   1:  PR[91,2] = PR[90,2] + -18.989;
   1:L PR[91] R[100]mm/sec CNT100;
   1:  PR[91,1] = PR[90,1] + -71.625;
   1:  PR[91,2] = PR[90,2] + -19.966;
   1:L PR[91] R[100]mm/sec CNT100;
   1:  PR[91,1] = PR[90,1] + -67.146;
   1:  PR[91,2] = PR[90,2] + -20.149;
   1:L PR[91] R[100]mm/sec CNT100;
   1:  PR[91,1] = PR[90,1] + -63.769;
   1:  PR[91,2] = PR[90,2] + -19.645;
   1:L PR[91] R[100]mm/sec CNT100;
   1:  PR[91,1] = PR[90,1] + -62.587;
   1:  PR[91,2] = PR[90,2] + -19.490;
   1:L PR[91] R[100]mm/sec CNT100;
   1:  PR[91,1] = PR[90,1] + -60.217;
   1:  PR[91,2] = PR[90,2] + -18.649;
   1:L PR[91] R[100]mm/sec CNT100;
   1:  PR[91,1] = PR[90,1] + -58.248;
   1:  PR[91,2] = PR[90,2] + -17.990;
   1:L PR[91] R[100]mm/sec CNT100;
   1:  PR[91,1] = PR[90,1] + -56.891;
   1:  PR[91,2] = PR[90,2] + -17.175;
   1:L PR[91] R[100]mm/sec CNT100;
   1:  PR[91,1] = PR[90,1] + -54.312;
   1:  PR[91,2] = PR[90,2] + -15.689;
   1:L PR[91] R[100]mm/sec CNT100;
   1:  PR[91,1] = PR[90,1] + -53.842;
   1:  PR[91,2] = PR[90,2] + -15.250;
   1:L PR[91] R[100]mm/sec CNT100;
   1:  PR[91,1] = PR[90,1] + -50.938;
   1:  PR[91,2] = PR[90,2] + -12.631;
   1:L PR[91] R[100]mm/sec CNT100;
   1:  PR[91,1] = PR[90,1] + -48.280;
   1:  PR[91,2] = PR[90,2] + -9.189;
   1:L PR[91] R[100]mm/sec CNT100TB   .50sec,CALL END_PUD;
   1:  PR[92] = PR[91];
   1:  PR[92,3] = PR[92,3] + 20;
   1:J PR[92] 10% FINE;
   1:  PR[91] = PR[90];
   1:  PR[91,1] = PR[90,1] + -47.207;
   1:  PR[91,2] = PR[90,2] + 7.658;
   1:  PR[91,3] = PR[90,3] + 39.195;
   1:  PR[92] = PR[91];
   1:  PR[92,3] = PR[92,3] + 20;
   1:J PR[92] 10% FINE;
   1:L PR[91] R[100]mm/sec CNT100;
   1:  CALL LASER_DRAHT_START;
   1:  PR[91,1] = PR[90,1] + -49.902;
   1:  PR[91,2] = PR[90,2] + 11.311;
   1:L PR[91] R[100]mm/sec CNT100;
   1:  PR[91,1] = PR[90,1] + -51.244;
   1:  PR[91,2] = PR[90,2] + 12.483;
   1:L PR[91] R[100]mm/sec CNT100;
   1:  PR[91,1] = PR[90,1] + -53.419;
   1:  PR[91,2] = PR[90,2] + 14.347;
   1:L PR[91] R[100]mm/sec CNT100;
   1:  PR[91,1] = PR[90,1] + -57.577;
   1:  PR[91,2] = PR[90,2] + 16.651;
   1:L PR[91] R[100]mm/sec CNT100;
   1:  PR[91,1] = PR[90,1] + -60.018;
   1:  PR[91,2] = PR[90,2] + 17.440;
   1:L PR[91] R[100]mm/sec CNT100;
   1:  PR[91,1] = PR[90,1] + -62.061;
   1:  PR[91,2] = PR[90,2] + 18.166;
   1:L PR[91] R[100]mm/sec CNT100;
   1:  PR[91,1] = PR[90,1] + -66.547;
   1:  PR[91,2] = PR[90,2] + 18.829;
   1:L PR[91] R[100]mm/sec CNT100;
   1:  PR[91,1] = PR[90,1] + -68.412;
   1:  PR[91,2] = PR[90,2] + 18.760;
   1:L PR[91] R[100]mm/sec CNT100;
   1:  PR[91,1] = PR[90,1] + -71.023;
   1:  PR[91,2] = PR[90,2] + 18.639;
   1:L PR[91] R[100]mm/sec CNT100;
   1:  PR[91,1] = PR[90,1] + -75.333;
   1:  PR[91,2] = PR[90,2] + 17.623;
   1:L PR[91] R[100]mm/sec CNT100;
   1:  PR[91,1] = PR[90,1] + -79.285;
   1:  PR[91,2] = PR[90,2] + 15.844;
   1:L PR[91] R[100]mm/sec CNT100;
   1:  PR[91,1] = PR[90,1] + -82.702;
   1:  PR[91,2] = PR[90,2] + 13.402;
   1:L PR[91] R[100]mm/sec CNT100;
   1:  PR[91,1] = PR[90,1] + -85.411;
   1:  PR[91,2] = PR[90,2] + 10.405;
   1:L PR[91] R[100]mm/sec CNT100;
   1:  PR[91,1] = PR[90,1] + -87.427;
   1:  PR[91,2] = PR[90,2] + 6.951;
   1:L PR[91] R[100]mm/sec CNT100;
   1:  PR[91,1] = PR[90,1] + -88.666;
   1:  PR[91,2] = PR[90,2] + 3.187;
   1:L PR[91] R[100]mm/sec CNT100;
   1:  PR[91,1] = PR[90,1] + -88.752;
   1:  PR[91,2] = PR[90,2] + 2.391;
   1:L PR[91] R[100]mm/sec CNT100;
   1:  PR[91,1] = PR[90,1] + -88.808;
   1:  PR[91,2] = PR[90,2] + 2.113;
   1:L PR[91] R[100]mm/sec CNT100;
   1:  PR[91,1] = PR[90,1] + -89.112;
   1:  PR[91,2] = PR[90,2] + -0.728;
   1:L PR[91] R[100]mm/sec CNT100;
   1:  PR[91,1] = PR[90,1] + -89.014;
   1:  PR[91,2] = PR[90,2] + -1.630;
   1:L PR[91] R[100]mm/sec CNT100;
   1:  PR[91,1] = PR[90,1] + -88.812;
   1:  PR[91,2] = PR[90,2] + -2.533;
   1:L PR[91] R[100]mm/sec CNT100;
   1:  PR[91,1] = PR[90,1] + -88.586;
   1:  PR[91,2] = PR[90,2] + -4.648;
   1:L PR[91] R[100]mm/sec CNT100;
   1:  PR[91,1] = PR[90,1] + -87.339;
   1:  PR[91,2] = PR[90,2] + -8.411;
   1:L PR[91] R[100]mm/sec CNT100;
   1:  PR[91,1] = PR[90,1] + -85.305;
   1:  PR[91,2] = PR[90,2] + -11.869;
   1:L PR[91] R[100]mm/sec CNT100;
   1:  PR[91,1] = PR[90,1] + -82.564;
   1:  PR[91,2] = PR[90,2] + -14.882;
   1:L PR[91] R[100]mm/sec CNT100;
   1:  PR[91,1] = PR[90,1] + -79.213;
   1:  PR[91,2] = PR[90,2] + -17.320;
   1:L PR[91] R[100]mm/sec CNT100;
   1:  PR[91,1] = PR[90,1] + -75.385;
   1:  PR[91,2] = PR[90,2] + -19.075;
   1:L PR[91] R[100]mm/sec CNT100;
   1:  PR[91,1] = PR[90,1] + -71.106;
   1:  PR[91,2] = PR[90,2] + -20.083;
   1:L PR[91] R[100]mm/sec CNT100;
   1:  PR[91,1] = PR[90,1] + -67.492;
   1:  PR[91,2] = PR[90,2] + -20.230;
   1:L PR[91] R[100]mm/sec CNT100;
   1:  PR[91,1] = PR[90,1] + -66.515;
   1:  PR[91,2] = PR[90,2] + -20.286;
   1:L PR[91] R[100]mm/sec CNT100;
   1:  PR[91,1] = PR[90,1] + -63.770;
   1:  PR[91,2] = PR[90,2] + -19.876;
   1:L PR[91] R[100]mm/sec CNT100;
   1:  PR[91,1] = PR[90,1] + -61.937;
   1:  PR[91,2] = PR[90,2] + -19.636;
   1:L PR[91] R[100]mm/sec CNT100;
   1:  PR[91,1] = PR[90,1] + -60.190;
   1:  PR[91,2] = PR[90,2] + -19.016;
   1:L PR[91] R[100]mm/sec CNT100;
   1:  PR[91,1] = PR[90,1] + -57.558;
   1:  PR[91,2] = PR[90,2] + -18.135;
   1:L PR[91] R[100]mm/sec CNT100;
   1:  PR[91,1] = PR[90,1] + -56.806;
   1:  PR[91,2] = PR[90,2] + -17.684;
   1:L PR[91] R[100]mm/sec CNT100;
   1:  PR[91,1] = PR[90,1] + -53.568;
   1:  PR[91,2] = PR[90,2] + -15.818;
   1:L PR[91] R[100]mm/sec CNT100;
   1:  PR[91,1] = PR[90,1] + -53.267;
   1:  PR[91,2] = PR[90,2] + -15.544;
   1:L PR[91] R[100]mm/sec CNT100;
   1:  PR[91,1] = PR[90,1] + -50.100;
   1:  PR[91,2] = PR[90,2] + -12.951;
   1:L PR[91] R[100]mm/sec CNT100;
   1:  PR[91,1] = PR[90,1] + -49.327;
   1:  PR[91,2] = PR[90,2] + -12.096;
   1:L PR[91] R[100]mm/sec CNT100;
   1:  PR[91,1] = PR[90,1] + -47.391;
   1:  PR[91,2] = PR[90,2] + -9.587;
   1:L PR[91] R[100]mm/sec CNT100;
   1:  PR[91,1] = PR[90,1] + -46.330;
   1:  PR[91,2] = PR[90,2] + -7.540;
   1:L PR[91] R[100]mm/sec CNT100;
   1:  PR[91,1] = PR[90,1] + -45.515;
   1:  PR[91,2] = PR[90,2] + -5.643;
   1:L PR[91] R[100]mm/sec CNT100;
   1:  PR[91,1] = PR[90,1] + -45.158;
   1:  PR[91,2] = PR[90,2] + -3.960;
   1:L PR[91] R[100]mm/sec CNT100;
   1:  PR[91,1] = PR[90,1] + -45.073;
   1:  PR[91,2] = PR[90,2] + -3.355;
   1:L PR[91] R[100]mm/sec CNT100;
   1:  PR[91,1] = PR[90,1] + -45.003;
   1:  PR[91,2] = PR[90,2] + -2.254;
   1:L PR[91] R[100]mm/sec CNT100;
   1:  PR[91,1] = PR[90,1] + -44.855;
   1:  PR[91,2] = PR[90,2] + -0.642;
   1:L PR[91] R[100]mm/sec CNT100;
   1:  PR[91,1] = PR[90,1] + -45.345;
   1:  PR[91,2] = PR[90,2] + 3.088;
   1:L PR[91] R[100]mm/sec CNT100;
   1:  PR[91,1] = PR[90,1] + -45.463;
   1:  PR[91,2] = PR[90,2] + 3.590;
   1:L PR[91] R[100]mm/sec CNT100;
   1:  PR[91,1] = PR[90,1] + -46.247;
   1:  PR[91,2] = PR[90,2] + 5.331;
   1:L PR[91] R[100]mm/sec CNT100;
   1:  PR[91,1] = PR[90,1] + -47.206;
   1:  PR[91,2] = PR[90,2] + 7.658;
   1:L PR[91] R[100]mm/sec CNT100TB   .50sec,CALL END_PUD;
   1:  PR[92] = PR[91];
   1:  PR[92,3] = PR[92,3] + 20;
   1:J PR[92] 10% FINE;
   1:  PR[91,1] = PR[90,1] + -40.199;
   1:  PR[91,2] = PR[90,2] + 4.341;
   1:  PR[92] = PR[91];
   1:  PR[92,3] = PR[92,3] + 20;
   1:J PR[92] 10% FINE;
   1:L PR[91] R[100]mm/sec CNT100;
   1:  CALL LASER_DRAHT_START;
   1:  PR[91,1] = PR[90,1] + -40.331;
   1:  PR[91,2] = PR[90,2] + 4.012;
   1:L PR[91] R[100]mm/sec CNT100;
   1:  PR[91,1] = PR[90,1] + -40.685;
   1:  PR[91,2] = PR[90,2] + 2.385;
   1:L PR[91] R[100]mm/sec CNT100;
   1:  PR[91,1] = PR[90,1] + -40.769;
   1:  PR[91,2] = PR[90,2] + 1.636;
   1:L PR[91] R[100]mm/sec CNT100;
   1:  PR[91,1] = PR[90,1] + -40.955;
   1:  PR[91,2] = PR[90,2] + -0.751;
   1:L PR[91] R[100]mm/sec CNT100;
   1:  PR[91,1] = PR[90,1] + -40.654;
   1:  PR[91,2] = PR[90,2] + -4.032;
   1:L PR[91] R[100]mm/sec CNT100;
   1:  PR[91,1] = PR[90,1] + -40.296;
   1:  PR[91,2] = PR[90,2] + -5.597;
   1:L PR[91] R[100]mm/sec CNT100;
   1:  PR[91,1] = PR[90,1] + -39.609;
   1:  PR[91,2] = PR[90,2] + -7.567;
   1:L PR[91] R[100]mm/sec CNT100;
   1:  PR[91,1] = PR[90,1] + -39.122;
   1:  PR[91,2] = PR[90,2] + -8.820;
   1:L PR[91] R[100]mm/sec CNT100;
   1:  PR[91,1] = PR[90,1] + -38.825;
   1:  PR[91,2] = PR[90,2] + -9.370;
   1:L PR[91] R[100]mm/sec CNT100;
   1:  PR[91,1] = PR[90,1] + -37.086;
   1:  PR[91,2] = PR[90,2] + -12.138;
   1:L PR[91] R[100]mm/sec CNT100;
   1:  PR[91,1] = PR[90,1] + -36.794;
   1:  PR[91,2] = PR[90,2] + -12.551;
   1:L PR[91] R[100]mm/sec CNT100;
   1:  PR[91,1] = PR[90,1] + -36.056;
   1:  PR[91,2] = PR[90,2] + -13.368;
   1:L PR[91] R[100]mm/sec CNT100;
   1:  PR[91,1] = PR[90,1] + -33.732;
   1:  PR[91,2] = PR[90,2] + -15.700;
   1:L PR[91] R[100]mm/sec CNT100;
   1:  PR[91,1] = PR[90,1] + -32.622;
   1:  PR[91,2] = PR[90,2] + -16.492;
   1:L PR[91] R[100]mm/sec CNT100;
   1:  PR[91,1] = PR[90,1] + -30.086;
   1:  PR[91,2] = PR[90,2] + -18.111;
   1:L PR[91] R[100]mm/sec CNT100;
   1:  PR[91,1] = PR[90,1] + -28.459;
   1:  PR[91,2] = PR[90,2] + -18.807;
   1:L PR[91] R[100]mm/sec CNT100;
   1:  PR[91,1] = PR[90,1] + -25.985;
   1:  PR[91,2] = PR[90,2] + -19.712;
   1:L PR[91] R[100]mm/sec CNT100;
   1:  PR[91,1] = PR[90,1] + -23.769;
   1:  PR[91,2] = PR[90,2] + -20.140;
   1:L PR[91] R[100]mm/sec CNT100;
   1:  PR[91,1] = PR[90,1] + -21.612;
   1:  PR[91,2] = PR[90,2] + -20.432;
   1:L PR[91] R[100]mm/sec CNT100;
   1:  PR[91,1] = PR[90,1] + -18.812;
   1:  PR[91,2] = PR[90,2] + -20.365;
   1:L PR[91] R[100]mm/sec CNT100;
   1:  PR[91,1] = PR[90,1] + -17.167;
   1:  PR[91,2] = PR[90,2] + -20.229;
   1:L PR[91] R[100]mm/sec CNT100;
   1:  PR[91,1] = PR[90,1] + -13.883;
   1:  PR[91,2] = PR[90,2] + -19.427;
   1:L PR[91] R[100]mm/sec CNT100;
   1:  PR[91,1] = PR[90,1] + -12.850;
   1:  PR[91,2] = PR[90,2] + -19.107;
   1:L PR[91] R[100]mm/sec CNT100;
   1:  PR[91,1] = PR[90,1] + -9.308;
   1:  PR[91,2] = PR[90,2] + -17.354;
   1:L PR[91] R[100]mm/sec CNT100;
   1:  PR[91,1] = PR[90,1] + -8.864;
   1:  PR[91,2] = PR[90,2] + -17.098;
   1:L PR[91] R[100]mm/sec CNT100;
   1:  PR[91,1] = PR[90,1] + -5.397;
   1:  PR[91,2] = PR[90,2] + -14.278;
   1:L PR[91] R[100]mm/sec CNT100;
   1:  PR[91,1] = PR[90,1] + -3.913;
   1:  PR[91,2] = PR[90,2] + -12.363;
   1:L PR[91] R[100]mm/sec CNT100;
   1:  PR[91,1] = PR[90,1] + -2.510;
   1:  PR[91,2] = PR[90,2] + -10.642;
   1:L PR[91] R[100]mm/sec CNT100;
   1:  PR[91,1] = PR[90,1] + -2.507;
   1:  PR[91,2] = PR[90,2] + -10.636;
   1:L PR[91] R[100]mm/sec CNT100;
   1:  PR[91,1] = PR[90,1] + -0.715;
   1:  PR[91,2] = PR[90,2] + -6.857;
   1:L PR[91] R[100]mm/sec CNT100;
   1:  PR[91,1] = PR[90,1] + -0.610;
   1:  PR[91,2] = PR[90,2] + -6.577;
   1:L PR[91] R[100]mm/sec CNT100;
   1:  PR[91,1] = PR[90,1] + 0.216;
   1:  PR[91,2] = PR[90,2] + -3.257;
   1:L PR[91] R[100]mm/sec CNT100;
   1:  PR[91,1] = PR[90,1] + 3.385;
   1:  PR[91,2] = PR[90,2] + -3.299;
   1:L PR[91] R[100]mm/sec CNT100;
   1:  PR[91,1] = PR[90,1] + 4.076;
   1:  PR[91,2] = PR[90,2] + -6.422;
   1:L PR[91] R[100]mm/sec CNT100;
   1:  PR[91,1] = PR[90,1] + 4.773;
   1:  PR[91,2] = PR[90,2] + -8.090;
   1:L PR[91] R[100]mm/sec CNT100;
   1:  PR[91,1] = PR[90,1] + 5.666;
   1:  PR[91,2] = PR[90,2] + -10.320;
   1:L PR[91] R[100]mm/sec CNT100;
   1:  PR[91,1] = PR[90,1] + 6.034;
   1:  PR[91,2] = PR[90,2] + -11.054;
   1:L PR[91] R[100]mm/sec CNT100;
   1:  PR[91,1] = PR[90,1] + 8.671;
   1:  PR[91,2] = PR[90,2] + -14.460;
   1:L PR[91] R[100]mm/sec CNT100;
   1:  PR[91,1] = PR[90,1] + 8.949;
   1:  PR[91,2] = PR[90,2] + -14.860;
   1:L PR[91] R[100]mm/sec CNT100;
   1:  PR[91,1] = PR[90,1] + 9.487;
   1:  PR[91,2] = PR[90,2] + -15.427;
   1:L PR[91] R[100]mm/sec CNT100;
   1:  PR[91,1] = PR[90,1] + 13.137;
   1:  PR[91,2] = PR[90,2] + -18.194;
   1:L PR[91] R[100]mm/sec CNT100;
   1:  PR[91,1] = PR[90,1] + 13.723;
   1:  PR[91,2] = PR[90,2] + -18.559;
   1:L PR[91] R[100]mm/sec CNT100;
   1:  PR[91,1] = PR[90,1] + 18.095;
   1:  PR[91,2] = PR[90,2] + -20.344;
   1:L PR[91] R[100]mm/sec CNT100;
   1:  PR[91,1] = PR[90,1] + 18.615;
   1:  PR[91,2] = PR[90,2] + -20.509;
   1:L PR[91] R[100]mm/sec CNT100;
   1:  PR[91,1] = PR[90,1] + 23.451;
   1:  PR[91,2] = PR[90,2] + -21.128;
   1:L PR[91] R[100]mm/sec CNT100;
   1:  PR[91,1] = PR[90,1] + 23.842;
   1:  PR[91,2] = PR[90,2] + -21.151;
   1:L PR[91] R[100]mm/sec CNT100;
   1:  PR[91,1] = PR[90,1] + 28.822;
   1:  PR[91,2] = PR[90,2] + -20.487;
   1:L PR[91] R[100]mm/sec CNT100;
   1:  PR[91,1] = PR[90,1] + 29.059;
   1:  PR[91,2] = PR[90,2] + -20.442;
   1:L PR[91] R[100]mm/sec CNT100;
   1:  PR[91,1] = PR[90,1] + 33.829;
   1:  PR[91,2] = PR[90,2] + -18.475;
   1:L PR[91] R[100]mm/sec CNT100;
   1:  PR[91,1] = PR[90,1] + 33.923;
   1:  PR[91,2] = PR[90,2] + -18.431;
   1:L PR[91] R[100]mm/sec CNT100;
   1:  PR[91,1] = PR[90,1] + 38.131;
   1:  PR[91,2] = PR[90,2] + -15.244;
   1:L PR[91] R[100]mm/sec CNT100;
   1:  PR[91,1] = PR[90,1] + 38.658;
   1:  PR[91,2] = PR[90,2] + -14.617;
   1:L PR[91] R[100]mm/sec CNT100;
   1:  PR[91,1] = PR[90,1] + 42.705;
   1:  PR[91,2] = PR[90,2] + -9.418;
   1:L PR[91] R[100]mm/sec CNT100;
   1:  PR[91,1] = PR[90,1] + 47.189;
   1:  PR[91,2] = PR[90,2] + -14.100;
   1:L PR[91] R[100]mm/sec CNT100;
   1:  PR[91,1] = PR[90,1] + 47.481;
   1:  PR[91,2] = PR[90,2] + -14.437;
   1:L PR[91] R[100]mm/sec CNT100;
   1:  PR[91,1] = PR[90,1] + 50.974;
   1:  PR[91,2] = PR[90,2] + -16.993;
   1:L PR[91] R[100]mm/sec CNT100;
   1:  PR[91,1] = PR[90,1] + 52.879;
   1:  PR[91,2] = PR[90,2] + -18.168;
   1:L PR[91] R[100]mm/sec CNT100;
   1:  PR[91,1] = PR[90,1] + 55.023;
   1:  PR[91,2] = PR[90,2] + -19.106;
   1:L PR[91] R[100]mm/sec CNT100;
   1:  PR[91,1] = PR[90,1] + 59.619;
   1:  PR[91,2] = PR[90,2] + -20.650;
   1:L PR[91] R[100]mm/sec CNT100;
   1:  PR[91,1] = PR[90,1] + 59.641;
   1:  PR[91,2] = PR[90,2] + -20.654;
   1:L PR[91] R[100]mm/sec CNT100;
   1:  PR[91,1] = PR[90,1] + 60.098;
   1:  PR[91,2] = PR[90,2] + -20.706;
   1:L PR[91] R[100]mm/sec CNT100;
   1:  PR[91,1] = PR[90,1] + 64.803;
   1:  PR[91,2] = PR[90,2] + -21.406;
   1:L PR[91] R[100]mm/sec CNT100;
   1:  PR[91,1] = PR[90,1] + 66.209;
   1:  PR[91,2] = PR[90,2] + -21.457;
   1:L PR[91] R[100]mm/sec CNT100;
   1:  PR[91,1] = PR[90,1] + 69.518;
   1:  PR[91,2] = PR[90,2] + -21.226;
   1:L PR[91] R[100]mm/sec CNT100;
   1:  PR[91,1] = PR[90,1] + 72.304;
   1:  PR[91,2] = PR[90,2] + -20.762;
   1:L PR[91] R[100]mm/sec CNT100;
   1:  PR[91,1] = PR[90,1] + 73.960;
   1:  PR[91,2] = PR[90,2] + -20.276;
   1:L PR[91] R[100]mm/sec CNT100;
   1:  PR[91,1] = PR[90,1] + 77.569;
   1:  PR[91,2] = PR[90,2] + -18.895;
   1:L PR[91] R[100]mm/sec CNT100;
   1:  PR[91,1] = PR[90,1] + 78.035;
   1:  PR[91,2] = PR[90,2] + -18.638;
   1:L PR[91] R[100]mm/sec CNT100;
   1:  PR[91,1] = PR[90,1] + 81.794;
   1:  PR[91,2] = PR[90,2] + -16.221;
   1:L PR[91] R[100]mm/sec CNT100;
   1:  PR[91,1] = PR[90,1] + 84.969;
   1:  PR[91,2] = PR[90,2] + -12.992;
   1:L PR[91] R[100]mm/sec CNT100;
   1:  PR[91,1] = PR[90,1] + 87.334;
   1:  PR[91,2] = PR[90,2] + -9.214;
   1:L PR[91] R[100]mm/sec CNT100;
   1:  PR[91,1] = PR[90,1] + 88.789;
   1:  PR[91,2] = PR[90,2] + -5.064;
   1:L PR[91] R[100]mm/sec CNT100;
   1:  PR[91,1] = PR[90,1] + 89.281;
   1:  PR[91,2] = PR[90,2] + -0.729;
   1:L PR[91] R[100]mm/sec CNT100;
   1:  PR[91,1] = PR[90,1] + 88.789;
   1:  PR[91,2] = PR[90,2] + 3.606;
   1:L PR[91] R[100]mm/sec CNT100;
   1:  PR[91,1] = PR[90,1] + 87.334;
   1:  PR[91,2] = PR[90,2] + 7.755;
   1:L PR[91] R[100]mm/sec CNT100;
   1:  PR[91,1] = PR[90,1] + 84.969;
   1:  PR[91,2] = PR[90,2] + 11.533;
   1:L PR[91] R[100]mm/sec CNT100;
   1:  PR[91,1] = PR[90,1] + 81.794;
   1:  PR[91,2] = PR[90,2] + 14.762;
   1:L PR[91] R[100]mm/sec CNT100;
   1:  PR[91,1] = PR[90,1] + 78.035;
   1:  PR[91,2] = PR[90,2] + 17.179;
   1:L PR[91] R[100]mm/sec CNT100;
   1:  PR[91,1] = PR[90,1] + 77.569;
   1:  PR[91,2] = PR[90,2] + 17.436;
   1:L PR[91] R[100]mm/sec CNT100;
   1:  PR[91,1] = PR[90,1] + 73.960;
   1:  PR[91,2] = PR[90,2] + 18.817;
   1:L PR[91] R[100]mm/sec CNT100;
   1:  PR[91,1] = PR[90,1] + 72.304;
   1:  PR[91,2] = PR[90,2] + 19.303;
   1:L PR[91] R[100]mm/sec CNT100;
   1:  PR[91,1] = PR[90,1] + 69.518;
   1:  PR[91,2] = PR[90,2] + 19.767;
   1:L PR[91] R[100]mm/sec CNT100;
   1:  PR[91,1] = PR[90,1] + 66.210;
   1:  PR[91,2] = PR[90,2] + 19.998;
   1:L PR[91] R[100]mm/sec CNT100;
   1:  PR[91,1] = PR[90,1] + 64.803;
   1:  PR[91,2] = PR[90,2] + 19.947;
   1:L PR[91] R[100]mm/sec CNT100;
   1:  PR[91,1] = PR[90,1] + 60.098;
   1:  PR[91,2] = PR[90,2] + 19.247;
   1:L PR[91] R[100]mm/sec CNT100;
   1:  PR[91,1] = PR[90,1] + 59.643;
   1:  PR[91,2] = PR[90,2] + 19.196;
   1:L PR[91] R[100]mm/sec CNT100;
   1:  PR[91,1] = PR[90,1] + 59.618;
   1:  PR[91,2] = PR[90,2] + 19.191;
   1:L PR[91] R[100]mm/sec CNT100;
   1:  PR[91,1] = PR[90,1] + 55.003;
   1:  PR[91,2] = PR[90,2] + 17.641;
   1:L PR[91] R[100]mm/sec CNT100;
   1:  PR[91,1] = PR[90,1] + 52.828;
   1:  PR[91,2] = PR[90,2] + 16.681;
   1:L PR[91] R[100]mm/sec CNT100;
   1:  PR[91,1] = PR[90,1] + 50.931;
   1:  PR[91,2] = PR[90,2] + 15.513;
   1:L PR[91] R[100]mm/sec CNT100;
   1:  PR[91,1] = PR[90,1] + 47.400;
   1:  PR[91,2] = PR[90,2] + 12.904;
   1:L PR[91] R[100]mm/sec CNT100;
   1:  PR[91,1] = PR[90,1] + 47.207;
   1:  PR[91,2] = PR[90,2] + 12.680;
   1:L PR[91] R[100]mm/sec CNT100;
   1:  PR[91,1] = PR[90,1] + 42.713;
   1:  PR[91,2] = PR[90,2] + 7.937;
   1:L PR[91] R[100]mm/sec CNT100;
   1:  PR[91,1] = PR[90,1] + 38.150;
   1:  PR[91,2] = PR[90,2] + 13.761;
   1:L PR[91] R[100]mm/sec CNT100;
   1:  PR[91,1] = PR[90,1] + 38.071;
   1:  PR[91,2] = PR[90,2] + 13.839;
   1:L PR[91] R[100]mm/sec CNT100;
   1:  PR[91,1] = PR[90,1] + 33.925;
   1:  PR[91,2] = PR[90,2] + 16.974;
   1:L PR[91] R[100]mm/sec CNT100;
   1:  PR[91,1] = PR[90,1] + 33.918;
   1:  PR[91,2] = PR[90,2] + 16.979;
   1:L PR[91] R[100]mm/sec CNT100;
   1:  PR[91,1] = PR[90,1] + 33.792;
   1:  PR[91,2] = PR[90,2] + 17.038;
   1:L PR[91] R[100]mm/sec CNT100;
   1:  PR[91,1] = PR[90,1] + 29.024;
   1:  PR[91,2] = PR[90,2] + 18.992;
   1:L PR[91] R[100]mm/sec CNT100;
   1:  PR[91,1] = PR[90,1] + 28.786;
   1:  PR[91,2] = PR[90,2] + 19.038;
   1:L PR[91] R[100]mm/sec CNT100;
   1:  PR[91,1] = PR[90,1] + 23.812;
   1:  PR[91,2] = PR[90,2] + 19.692;
   1:L PR[91] R[100]mm/sec CNT100;
   1:  PR[91,1] = PR[90,1] + 23.421;
   1:  PR[91,2] = PR[90,2] + 19.670;
   1:L PR[91] R[100]mm/sec CNT100;
   1:  PR[91,1] = PR[90,1] + 18.592;
   1:  PR[91,2] = PR[90,2] + 19.044;
   1:L PR[91] R[100]mm/sec CNT100;
   1:  PR[91,1] = PR[90,1] + 18.072;
   1:  PR[91,2] = PR[90,2] + 18.880;
   1:L PR[91] R[100]mm/sec CNT100;
   1:  PR[91,1] = PR[90,1] + 13.707;
   1:  PR[91,2] = PR[90,2] + 17.092;
   1:L PR[91] R[100]mm/sec CNT100;
   1:  PR[91,1] = PR[90,1] + 13.121;
   1:  PR[91,2] = PR[90,2] + 16.727;
   1:L PR[91] R[100]mm/sec CNT100;
   1:  PR[91,1] = PR[90,1] + 9.478;
   1:  PR[91,2] = PR[90,2] + 13.959;
   1:L PR[91] R[100]mm/sec CNT100;
   1:  PR[91,1] = PR[90,1] + 8.904;
   1:  PR[91,2] = PR[90,2] + 13.356;
   1:L PR[91] R[100]mm/sec CNT100;
   1:  PR[91,1] = PR[90,1] + 6.144;
   1:  PR[91,2] = PR[90,2] + 9.789;
   1:L PR[91] R[100]mm/sec CNT100;
   1:  PR[91,1] = PR[90,1] + 6.104;
   1:  PR[91,2] = PR[90,2] + 9.727;
   1:L PR[91] R[100]mm/sec CNT100;
   1:  PR[91,1] = PR[90,1] + 5.769;
   1:  PR[91,2] = PR[90,2] + 9.085;
   1:L PR[91] R[100]mm/sec CNT100;
   1:  PR[91,1] = PR[90,1] + 4.383;
   1:  PR[91,2] = PR[90,2] + 5.768;
   1:L PR[91] R[100]mm/sec CNT100;
   1:  PR[91,1] = PR[90,1] + 4.103;
   1:  PR[91,2] = PR[90,2] + 5.061;
   1:L PR[91] R[100]mm/sec CNT100;
   1:  PR[91,1] = PR[90,1] + 3.380;
   1:  PR[91,2] = PR[90,2] + 1.835;
   1:L PR[91] R[100]mm/sec CNT100;
   1:  PR[91,1] = PR[90,1] + 0.218;
   1:  PR[91,2] = PR[90,2] + 1.796;
   1:L PR[91] R[100]mm/sec CNT100;
   1:  PR[91,1] = PR[90,1] + -0.605;
   1:  PR[91,2] = PR[90,2] + 5.086;
   1:L PR[91] R[100]mm/sec CNT100;
   1:  PR[91,1] = PR[90,1] + -2.193;
   1:  PR[91,2] = PR[90,2] + 8.477;
   1:L PR[91] R[100]mm/sec CNT100;
   1:  PR[91,1] = PR[90,1] + -2.509;
   1:  PR[91,2] = PR[90,2] + 9.179;
   1:L PR[91] R[100]mm/sec CNT100;
   1:  PR[91,1] = PR[90,1] + -3.914;
   1:  PR[91,2] = PR[90,2] + 10.905;
   1:L PR[91] R[100]mm/sec CNT100;
   1:  PR[91,1] = PR[90,1] + -5.385;
   1:  PR[91,2] = PR[90,2] + 12.808;
   1:L PR[91] R[100]mm/sec CNT100;
   1:  PR[91,1] = PR[90,1] + -8.852;
   1:  PR[91,2] = PR[90,2] + 15.632;
   1:L PR[91] R[100]mm/sec CNT100;
   1:  PR[91,1] = PR[90,1] + -9.296;
   1:  PR[91,2] = PR[90,2] + 15.887;
   1:L PR[91] R[100]mm/sec CNT100;
   1:  PR[91,1] = PR[90,1] + -12.840;
   1:  PR[91,2] = PR[90,2] + 17.644;
   1:L PR[91] R[100]mm/sec CNT100;
   1:  PR[91,1] = PR[90,1] + -13.871;
   1:  PR[91,2] = PR[90,2] + 17.964;
   1:L PR[91] R[100]mm/sec CNT100;
   1:  PR[91,1] = PR[90,1] + -17.158;
   1:  PR[91,2] = PR[90,2] + 18.769;
   1:L PR[91] R[100]mm/sec CNT100;
   1:  PR[91,1] = PR[90,1] + -18.802;
   1:  PR[91,2] = PR[90,2] + 18.905;
   1:L PR[91] R[100]mm/sec CNT100;
   1:  PR[91,1] = PR[90,1] + -21.605;
   1:  PR[91,2] = PR[90,2] + 18.974;
   1:L PR[91] R[100]mm/sec CNT100;
   1:  PR[91,1] = PR[90,1] + -23.761;
   1:  PR[91,2] = PR[90,2] + 18.682;
   1:L PR[91] R[100]mm/sec CNT100;
   1:  PR[91,1] = PR[90,1] + -25.979;
   1:  PR[91,2] = PR[90,2] + 18.255;
   1:L PR[91] R[100]mm/sec CNT100;
   1:  PR[91,1] = PR[90,1] + -28.453;
   1:  PR[91,2] = PR[90,2] + 17.350;
   1:L PR[91] R[100]mm/sec CNT100;
   1:  PR[91,1] = PR[90,1] + -30.082;
   1:  PR[91,2] = PR[90,2] + 16.654;
   1:L PR[91] R[100]mm/sec CNT100;
   1:  PR[91,1] = PR[90,1] + -32.618;
   1:  PR[91,2] = PR[90,2] + 15.035;
   1:L PR[91] R[100]mm/sec CNT100;
   1:  PR[91,1] = PR[90,1] + -33.730;
   1:  PR[91,2] = PR[90,2] + 14.244;
   1:L PR[91] R[100]mm/sec CNT100;
   1:  PR[91,1] = PR[90,1] + -36.054;
   1:  PR[91,2] = PR[90,2] + 11.911;
   1:L PR[91] R[100]mm/sec CNT100;
   1:  PR[91,1] = PR[90,1] + -36.756;
   1:  PR[91,2] = PR[90,2] + 11.135;
   1:L PR[91] R[100]mm/sec CNT100;
   1:  PR[91,1] = PR[90,1] + -38.708;
   1:  PR[91,2] = PR[90,2] + 8.037;
   1:L PR[91] R[100]mm/sec CNT100;
   1:  PR[91,1] = PR[90,1] + -38.832;
   1:  PR[91,2] = PR[90,2] + 7.886;
   1:L PR[91] R[100]mm/sec CNT100;
   1:  PR[91,1] = PR[90,1] + -38.946;
   1:  PR[91,2] = PR[90,2] + 7.712;
   1:L PR[91] R[100]mm/sec CNT100;
   1:  PR[91,1] = PR[90,1] + -39.077;
   1:  PR[91,2] = PR[90,2] + 7.458;
   1:L PR[91] R[100]mm/sec CNT100;
   1:  PR[91,1] = PR[90,1] + -40.128;
   1:  PR[91,2] = PR[90,2] + 4.457;
   1:L PR[91] R[100]mm/sec CNT100;
   1:  PR[91,1] = PR[90,1] + -40.199;
   1:  PR[91,2] = PR[90,2] + 4.341;
   1:L PR[91] R[100]mm/sec CNT100TB   .50sec,CALL END_PUD;
   1:  PR[92] = PR[91];
   1:  PR[92,3] = PR[92,3] + 20;
   1:J PR[92] 10% FINE;
   1:  PR[91] = PR[90];
   1:  PR[91,1] = PR[90,1] + -65.992;
   1:  PR[91,2] = PR[90,2] + 18.957;
   1:  PR[91,3] = PR[90,3] + 40.495;
   1:  PR[92] = PR[91];
   1:  PR[92,3] = PR[92,3] + 20;
   1:J PR[92] 10% FINE;
   1:L PR[91] R[100]mm/sec CNT100;
   1:  CALL LASER_DRAHT_START;
   1:  PR[91,1] = PR[90,1] + -70.510;
   1:  PR[91,2] = PR[90,2] + 18.756;
   1:L PR[91] R[100]mm/sec CNT100;
   1:  PR[91,1] = PR[90,1] + -72.599;
   1:  PR[91,2] = PR[90,2] + 18.270;
   1:  PR[91,3] = PR[90,3] + 39.207;
   1:L PR[91] R[100]mm/sec CNT100;
   1:  PR[91,1] = PR[90,1] + -74.831;
   1:  PR[91,2] = PR[90,2] + 17.729;
   1:  PR[91,3] = PR[90,3] + 39.213;
   1:L PR[91] R[100]mm/sec CNT100;
   1:  PR[91,1] = PR[90,1] + -78.808;
   1:  PR[91,2] = PR[90,2] + 15.932;
   1:  PR[91,3] = PR[90,3] + 39.219;
   1:L PR[91] R[100]mm/sec CNT100;
   1:  PR[91,1] = PR[90,1] + -82.272;
   1:  PR[91,2] = PR[90,2] + 13.461;
   1:  PR[91,3] = PR[90,3] + 39.231;
   1:L PR[91] R[100]mm/sec CNT100;
   1:  PR[91,1] = PR[90,1] + -85.098;
   1:  PR[91,2] = PR[90,2] + 10.424;
   1:  PR[91,3] = PR[90,3] + 39.243;
   1:L PR[91] R[100]mm/sec CNT100;
   1:  PR[91,1] = PR[90,1] + -85.488;
   1:  PR[91,2] = PR[90,2] + 9.776;
   1:  PR[91,3] = PR[90,3] + 39.254;
   1:L PR[91] R[100]mm/sec CNT100;
   1:  PR[91,1] = PR[90,1] + -87.119;
   1:  PR[91,2] = PR[90,2] + 6.978;
   1:  PR[91,3] = PR[90,3] + 39.256;
   1:L PR[91] R[100]mm/sec CNT100;
   1:  PR[91,1] = PR[90,1] + -88.368;
   1:  PR[91,2] = PR[90,2] + 3.180;
   1:  PR[91,3] = PR[90,3] + 39.265;
   1:L PR[91] R[100]mm/sec CNT100;
   1:  PR[91,1] = PR[90,1] + -88.408;
   1:  PR[91,2] = PR[90,2] + 2.869;
   1:  PR[91,3] = PR[90,3] + 39.276;
   1:L PR[91] R[100]mm/sec CNT100;
   1:  PR[91,1] = PR[90,1] + -88.794;
   1:  PR[91,2] = PR[90,2] + -0.728;
   1:  PR[91,3] = PR[90,3] + 39.277;
   1:L PR[91] R[100]mm/sec CNT100;
   1:  PR[91,1] = PR[90,1] + -88.766;
   1:  PR[91,2] = PR[90,2] + -0.984;
   1:  PR[91,3] = PR[90,3] + 39.286;
   1:L PR[91] R[100]mm/sec CNT100;
   1:  PR[91,1] = PR[90,1] + -88.520;
   1:  PR[91,2] = PR[90,2] + -2.078;
   1:  PR[91,3] = PR[90,3] + 39.287;
   1:L PR[91] R[100]mm/sec CNT100;
   1:  PR[91,1] = PR[90,1] + -88.244;
   1:  PR[91,2] = PR[90,2] + -4.663;
   1:  PR[91,3] = PR[90,3] + 39.290;
   1:L PR[91] R[100]mm/sec CNT100;
   1:  PR[91,1] = PR[90,1] + -86.993;
   1:  PR[91,2] = PR[90,2] + -8.441;
   1:  PR[91,3] = PR[90,3] + 39.297;
   1:L PR[91] R[100]mm/sec CNT100;
   1:  PR[91,1] = PR[90,1] + -84.954;
   1:  PR[91,2] = PR[90,2] + -11.914;
   1:  PR[91,3] = PR[90,3] + 39.308;
   1:L PR[91] R[100]mm/sec CNT100;
   1:  PR[91,1] = PR[90,1] + -82.204;
   1:  PR[91,2] = PR[90,2] + -14.942;
   1:  PR[91,3] = PR[90,3] + 39.319;
   1:L PR[91] R[100]mm/sec CNT100;
   1:  PR[91,1] = PR[90,1] + -78.842;
   1:  PR[91,2] = PR[90,2] + -17.393;
   1:  PR[91,3] = PR[90,3] + 39.330;
   1:L PR[91] R[100]mm/sec CNT100;
   1:  PR[91,1] = PR[90,1] + -76.437;
   1:  PR[91,2] = PR[90,2] + -18.498;
   1:  PR[91,3] = PR[90,3] + 39.341;
   1:L PR[91] R[100]mm/sec CNT100;
   1:  PR[91,1] = PR[90,1] + -74.938;
   1:  PR[91,2] = PR[90,2] + -19.169;
   1:  PR[91,3] = PR[90,3] + 39.349;
   1:L PR[91] R[100]mm/sec CNT100;
   1:  PR[91,1] = PR[90,1] + -71.259;
   1:  PR[91,2] = PR[90,2] + -20.025;
   1:  PR[91,3] = PR[90,3] + 39.353;
   1:L PR[91] R[100]mm/sec CNT100;
   1:  PR[91,1] = PR[90,1] + -70.510;
   1:  PR[91,2] = PR[90,2] + -20.211;
   1:  PR[91,3] = PR[90,3] + 39.363;
   1:L PR[91] R[100]mm/sec CNT100;
   1:  PR[91,1] = PR[90,1] + -67.495;
   1:  PR[91,2] = PR[90,2] + -20.334;
   1:  PR[91,3] = PR[90,3] + 39.365;
   1:L PR[91] R[100]mm/sec CNT100;
   1:  PR[91,1] = PR[90,1] + -65.902;
   1:  PR[91,2] = PR[90,2] + -20.425;
   1:  PR[91,3] = PR[90,3] + 39.374;
   1:L PR[91] R[100]mm/sec CNT100;
   1:  PR[91,1] = PR[90,1] + -63.771;
   1:  PR[91,2] = PR[90,2] + -20.108;
   1:  PR[91,3] = PR[90,3] + 39.378;
   1:L PR[91] R[100]mm/sec CNT100;
   1:  PR[91,1] = PR[90,1] + -61.287;
   1:  PR[91,2] = PR[90,2] + -19.782;
   1:  PR[91,3] = PR[90,3] + 39.384;
   1:L PR[91] R[100]mm/sec CNT100;
   1:  PR[91,1] = PR[90,1] + -60.163;
   1:  PR[91,2] = PR[90,2] + -19.383;
   1:  PR[91,3] = PR[90,3] + 39.391;
   1:L PR[91] R[100]mm/sec CNT100;
   1:  PR[91,1] = PR[90,1] + -56.854;
   1:  PR[91,2] = PR[90,2] + -18.276;
   1:  PR[91,3] = PR[90,3] + 39.394;
   1:L PR[91] R[100]mm/sec CNT100;
   1:  PR[91,1] = PR[90,1] + -55.345;
   1:  PR[91,2] = PR[90,2] + -17.399;
   1:  PR[91,3] = PR[90,3] + 39.403;
   1:L PR[91] R[100]mm/sec CNT100;
   1:  PR[91,1] = PR[90,1] + -52.784;
   1:  PR[91,2] = PR[90,2] + -16.071;
   1:  PR[91,3] = PR[90,3] + 39.408;
   1:L PR[91] R[100]mm/sec CNT100;
   1:  PR[91,1] = PR[90,1] + -52.031;
   1:  PR[91,2] = PR[90,2] + -15.552;
   1:  PR[91,3] = PR[90,3] + 39.416;
   1:L PR[91] R[100]mm/sec CNT100;
   1:  PR[91,1] = PR[90,1] + -49.353;
   1:  PR[91,2] = PR[90,2] + -13.360;
   1:  PR[91,3] = PR[90,3] + 39.418;
   1:L PR[91] R[100]mm/sec CNT100;
   1:  PR[91,1] = PR[90,1] + -47.673;
   1:  PR[91,2] = PR[90,2] + -11.503;
   1:  PR[91,3] = PR[90,3] + 39.428;
   1:L PR[91] R[100]mm/sec CNT100;
   1:  PR[91,1] = PR[90,1] + -46.502;
   1:  PR[91,2] = PR[90,2] + -9.984;
   1:  PR[91,3] = PR[90,3] + 39.435;
   1:L PR[91] R[100]mm/sec CNT100;
   1:  PR[91,1] = PR[90,1] + -44.819;
   1:  PR[91,2] = PR[90,2] + -6.737;
   1:  PR[91,3] = PR[90,3] + 39.440;
   1:L PR[91] R[100]mm/sec CNT100;
   1:  PR[91,1] = PR[90,1] + -44.494;
   1:  PR[91,2] = PR[90,2] + -5.982;
   1:  PR[91,3] = PR[90,3] + 39.450;
   1:L PR[91] R[100]mm/sec CNT100;
   1:  PR[91,1] = PR[90,1] + -43.886;
   1:  PR[91,2] = PR[90,2] + -3.116;
   1:  PR[91,3] = PR[90,3] + 39.452;
   1:L PR[91] R[100]mm/sec CNT100;
   1:  PR[91,1] = PR[90,1] + -40.672;
   1:  PR[91,2] = PR[90,2] + -3.090;
   1:  PR[91,3] = PR[90,3] + 39.460;
   1:L PR[91] R[100]mm/sec CNT100;
   1:  PR[91,1] = PR[90,1] + -40.009;
   1:  PR[91,2] = PR[90,2] + -5.989;
   1:  PR[91,3] = PR[90,3] + 39.469;
   1:L PR[91] R[100]mm/sec CNT100;
   1:  PR[91,1] = PR[90,1] + -39.713;
   1:  PR[91,2] = PR[90,2] + -6.837;
   1:  PR[91,3] = PR[90,3] + 39.477;
   1:L PR[91] R[100]mm/sec CNT100;
   1:  PR[91,1] = PR[90,1] + -38.974;
   1:  PR[91,2] = PR[90,2] + -8.740;
   1:  PR[91,3] = PR[90,3] + 39.479;
   1:L PR[91] R[100]mm/sec CNT100;
   1:  PR[91,1] = PR[90,1] + -38.498;
   1:  PR[91,2] = PR[90,2] + -9.622;
   1:  PR[91,3] = PR[90,3] + 39.485;
   1:L PR[91] R[100]mm/sec CNT100;
   1:  PR[91,1] = PR[90,1] + -37.059;
   1:  PR[91,2] = PR[90,2] + -11.912;
   1:  PR[91,3] = PR[90,3] + 39.487;
   1:L PR[91] R[100]mm/sec CNT100;
   1:  PR[91,1] = PR[90,1] + -36.612;
   1:  PR[91,2] = PR[90,2] + -12.544;
   1:  PR[91,3] = PR[90,3] + 39.495;
   1:L PR[91] R[100]mm/sec CNT100;
   1:  PR[91,1] = PR[90,1] + -35.538;
   1:  PR[91,2] = PR[90,2] + -13.733;
   1:  PR[91,3] = PR[90,3] + 39.497;
   1:L PR[91] R[100]mm/sec CNT100;
   1:  PR[91,1] = PR[90,1] + -33.554;
   1:  PR[91,2] = PR[90,2] + -15.725;
   1:  PR[91,3] = PR[90,3] + 39.501;
   1:L PR[91] R[100]mm/sec CNT100;
   1:  PR[91,1] = PR[90,1] + -32.019;
   1:  PR[91,2] = PR[90,2] + -16.819;
   1:  PR[91,3] = PR[90,3] + 39.509;
   1:L PR[91] R[100]mm/sec CNT100;
   1:  PR[91,1] = PR[90,1] + -29.908;
   1:  PR[91,2] = PR[90,2] + -18.167;
   1:  PR[91,3] = PR[90,3] + 39.514;
   1:L PR[91] R[100]mm/sec CNT100;
   1:  PR[91,1] = PR[90,1] + -27.776;
   1:  PR[91,2] = PR[90,2] + -19.079;
   1:  PR[91,3] = PR[90,3] + 39.521;
   1:L PR[91] R[100]mm/sec CNT100;
   1:  PR[91,1] = PR[90,1] + -25.799;
   1:  PR[91,2] = PR[90,2] + -19.802;
   1:  PR[91,3] = PR[90,3] + 39.527;
   1:L PR[91] R[100]mm/sec CNT100;
   1:  PR[91,1] = PR[90,1] + -23.017;
   1:  PR[91,2] = PR[90,2] + -20.339;
   1:  PR[91,3] = PR[90,3] + 39.533;
   1:L PR[91] R[100]mm/sec CNT100;
   1:  PR[91,1] = PR[90,1] + -21.413;
   1:  PR[91,2] = PR[90,2] + -20.557;
   1:  PR[91,3] = PR[90,3] + 39.541;
   1:L PR[91] R[100]mm/sec CNT100;
   1:  PR[91,1] = PR[90,1] + -18.007;
   1:  PR[91,2] = PR[90,2] + -20.475;
   1:  PR[91,3] = PR[90,3] + 39.545;
   1:L PR[91] R[100]mm/sec CNT100;
   1:  PR[91,1] = PR[90,1] + -16.945;
   1:  PR[91,2] = PR[90,2] + -20.387;
   1:  PR[91,3] = PR[90,3] + 39.554;
   1:L PR[91] R[100]mm/sec CNT100;
   1:  PR[91,1] = PR[90,1] + -13.047;
   1:  PR[91,2] = PR[90,2] + -19.435;
   1:  PR[91,3] = PR[90,3] + 39.557;
   1:L PR[91] R[100]mm/sec CNT100;
   1:  PR[91,1] = PR[90,1] + -12.597;
   1:  PR[91,2] = PR[90,2] + -19.296;
   1:  PR[91,3] = PR[90,3] + 39.568;
   1:L PR[91] R[100]mm/sec CNT100;
   1:  PR[91,1] = PR[90,1] + -8.520;
   1:  PR[91,2] = PR[90,2] + -17.271;
   1:  PR[91,3] = PR[90,3] + 39.569;
   1:L PR[91] R[100]mm/sec CNT100;
   1:  PR[91,1] = PR[90,1] + -7.905;
   1:  PR[91,2] = PR[90,2] + -16.771;
   1:  PR[91,3] = PR[90,3] + 39.582;
   1:L PR[91] R[100]mm/sec CNT100;
   1:  PR[91,1] = PR[90,1] + -4.834;
   1:  PR[91,2] = PR[90,2] + -14.411;
   1:  PR[91,3] = PR[90,3] + 39.584;
   1:L PR[91] R[100]mm/sec CNT100;
   1:  PR[91,1] = PR[90,1] + -4.616;
   1:  PR[91,2] = PR[90,2] + -14.178;
   1:  PR[91,3] = PR[90,3] + 39.594;
   1:L PR[91] R[100]mm/sec CNT100;
   1:  PR[91,1] = PR[90,1] + -1.952;
   1:  PR[91,2] = PR[90,2] + -10.910;
   1:  PR[91,3] = PR[90,3] + 39.595;
   1:L PR[91] R[100]mm/sec CNT100;
   1:  PR[91,1] = PR[90,1] + -1.574;
   1:  PR[91,2] = PR[90,2] + -10.195;
   1:  PR[91,3] = PR[90,3] + 39.607;
   1:L PR[91] R[100]mm/sec CNT100;
   1:  PR[91,1] = PR[90,1] + -0.351;
   1:  PR[91,2] = PR[90,2] + -7.616;
   1:  PR[91,3] = PR[90,3] + 39.609;
   1:L PR[91] R[100]mm/sec CNT100;
   1:  PR[91,1] = PR[90,1] + -0.010;
   1:  PR[91,2] = PR[90,2] + -6.708;
   1:  PR[91,3] = PR[90,3] + 39.617;
   1:L PR[91] R[100]mm/sec CNT100;
   1:  PR[91,1] = PR[90,1] + 0.373;
   1:  PR[91,2] = PR[90,2] + -5.172;
   1:  PR[91,3] = PR[90,3] + 39.619;
   1:L PR[91] R[100]mm/sec CNT100;
   1:  PR[91,1] = PR[90,1] + 3.542;
   1:  PR[91,2] = PR[90,2] + -5.213;
   1:  PR[91,3] = PR[90,3] + 39.624;
   1:L PR[91] R[100]mm/sec CNT100;
   1:  PR[91,1] = PR[90,1] + 3.871;
   1:  PR[91,2] = PR[90,2] + -6.703;
   1:  PR[91,3] = PR[90,3] + 39.632;
   1:L PR[91] R[100]mm/sec CNT100;
   1:  PR[91,1] = PR[90,1] + 5.193;
   1:  PR[91,2] = PR[90,2] + -9.999;
   1:  PR[91,3] = PR[90,3] + 39.636;
   1:L PR[91] R[100]mm/sec CNT100;
   1:  PR[91,1] = PR[90,1] + 5.803;
   1:  PR[91,2] = PR[90,2] + -11.215;
   1:  PR[91,3] = PR[90,3] + 39.646;
   1:L PR[91] R[100]mm/sec CNT100;
   1:  PR[91,1] = PR[90,1] + 8.008;
   1:  PR[91,2] = PR[90,2] + -14.064;
   1:  PR[91,3] = PR[90,3] + 39.650;
   1:L PR[91] R[100]mm/sec CNT100;
   1:  PR[91,1] = PR[90,1] + 8.465;
   1:  PR[91,2] = PR[90,2] + -14.721;
   1:  PR[91,3] = PR[90,3] + 39.659;
   1:L PR[91] R[100]mm/sec CNT100;
   1:  PR[91,1] = PR[90,1] + 9.404;
   1:  PR[91,2] = PR[90,2] + -15.711;
   1:  PR[91,3] = PR[90,3] + 39.662;
   1:L PR[91] R[100]mm/sec CNT100;
   1:  PR[91,1] = PR[90,1] + 12.621;
   1:  PR[91,2] = PR[90,2] + -18.150;
   1:  PR[91,3] = PR[90,3] + 39.665;
   1:L PR[91] R[100]mm/sec CNT100;
   1:  PR[91,1] = PR[90,1] + 13.690;
   1:  PR[91,2] = PR[90,2] + -18.816;
   1:  PR[91,3] = PR[90,3] + 39.676;
   1:L PR[91] R[100]mm/sec CNT100;
   1:  PR[91,1] = PR[90,1] + 17.565;
   1:  PR[91,2] = PR[90,2] + -20.398;
   1:  PR[91,3] = PR[90,3] + 39.680;
   1:L PR[91] R[100]mm/sec CNT100;
   1:  PR[91,1] = PR[90,1] + 18.622;
   1:  PR[91,2] = PR[90,2] + -20.733;
   1:  PR[91,3] = PR[90,3] + 39.691;
   1:L PR[91] R[100]mm/sec CNT100;
   1:  PR[91,1] = PR[90,1] + 22.930;
   1:  PR[91,2] = PR[90,2] + -21.284;
   1:  PR[91,3] = PR[90,3] + 39.694;
   1:L PR[91] R[100]mm/sec CNT100;
   1:  PR[91,1] = PR[90,1] + 23.878;
   1:  PR[91,2] = PR[90,2] + -21.339;
   1:  PR[91,3] = PR[90,3] + 39.706;
   1:L PR[91] R[100]mm/sec CNT100;
   1:  PR[91,1] = PR[90,1] + 28.337;
   1:  PR[91,2] = PR[90,2] + -20.745;
   1:  PR[91,3] = PR[90,3] + 39.708;
   1:L PR[91] R[100]mm/sec CNT100;
   1:  PR[91,1] = PR[90,1] + 29.114;
   1:  PR[91,2] = PR[90,2] + -20.594;
   1:  PR[91,3] = PR[90,3] + 39.721;
   1:L PR[91] R[100]mm/sec CNT100;
   1:  PR[91,1] = PR[90,1] + 33.406;
   1:  PR[91,2] = PR[90,2] + -18.825;
   1:  PR[91,3] = PR[90,3] + 39.723;
   1:L PR[91] R[100]mm/sec CNT100;
   1:  PR[91,1] = PR[90,1] + 33.989;
   1:  PR[91,2] = PR[90,2] + -18.551;
   1:  PR[91,3] = PR[90,3] + 39.735;
   1:L PR[91] R[100]mm/sec CNT100;
   1:  PR[91,1] = PR[90,1] + 37.880;
   1:  PR[91,2] = PR[90,2] + -15.598;
   1:  PR[91,3] = PR[90,3] + 39.737;
   1:L PR[91] R[100]mm/sec CNT100;
   1:  PR[91,1] = PR[90,1] + 37.983;
   1:  PR[91,2] = PR[90,2] + -15.533;
   1:  PR[91,3] = PR[90,3] + 39.750;
   1:L PR[91] R[100]mm/sec CNT100;
   1:  PR[91,1] = PR[90,1] + 38.302;
   1:  PR[91,2] = PR[90,2] + -15.236;
   1:  PR[91,3] = PR[90,3] + 39.751;
   1:L PR[91] R[100]mm/sec CNT100;
   1:  PR[91,1] = PR[90,1] + 38.533;
   1:  PR[91,2] = PR[90,2] + -14.984;
   1:  PR[91,3] = PR[90,3] + 39.752;
   1:L PR[91] R[100]mm/sec CNT100;
   1:  PR[91,1] = PR[90,1] + 40.180;
   1:  PR[91,2] = PR[90,2] + -12.996;
   1:  PR[91,3] = PR[90,3] + 39.753;
   1:L PR[91] R[100]mm/sec CNT100;
   1:  PR[91,1] = PR[90,1] + 42.121;
   1:  PR[91,2] = PR[90,2] + -10.502;
   1:  PR[91,3] = PR[90,3] + 39.760;
   1:L PR[91] R[100]mm/sec CNT100;
   1:  PR[91,1] = PR[90,1] + 44.418;
   1:  PR[91,2] = PR[90,2] + -12.906;
   1:  PR[91,3] = PR[90,3] + 39.768;
   1:L PR[91] R[100]mm/sec CNT100;
   1:  PR[91,1] = PR[90,1] + 45.836;
   1:  PR[91,2] = PR[90,2] + -14.345;
   1:  PR[91,3] = PR[90,3] + 39.778;
   1:L PR[91] R[100]mm/sec CNT100;
   1:  PR[91,1] = PR[90,1] + 46.719;
   1:  PR[91,2] = PR[90,2] + -14.975;
   1:  PR[91,3] = PR[90,3] + 39.783;
   1:L PR[91] R[100]mm/sec CNT100;
   1:  PR[91,1] = PR[90,1] + 48.779;
   1:  PR[91,2] = PR[90,2] + -16.323;
   1:  PR[91,3] = PR[90,3] + 39.786;
   1:L PR[91] R[100]mm/sec CNT100;
   1:  PR[91,1] = PR[90,1] + 50.613;
   1:  PR[91,2] = PR[90,2] + -17.665;
   1:  PR[91,3] = PR[90,3] + 39.793;
   1:L PR[91] R[100]mm/sec CNT100;
   1:  PR[91,1] = PR[90,1] + 51.361;
   1:  PR[91,2] = PR[90,2] + -18.127;
   1:  PR[91,3] = PR[90,3] + 39.799;
   1:L PR[91] R[100]mm/sec CNT100;
   1:  PR[91,1] = PR[90,1] + 54.713;
   1:  PR[91,2] = PR[90,2] + -19.592;
   1:  PR[91,3] = PR[90,3] + 39.801;
   1:L PR[91] R[100]mm/sec CNT100;
   1:  PR[91,1] = PR[90,1] + 58.060;
   1:  PR[91,2] = PR[90,2] + -20.717;
   1:  PR[91,3] = PR[90,3] + 39.811;
   1:L PR[91] R[100]mm/sec CNT100;
   1:  PR[91,1] = PR[90,1] + 59.336;
   1:  PR[91,2] = PR[90,2] + -20.988;
   1:  PR[91,3] = PR[90,3] + 39.821;
   1:L PR[91] R[100]mm/sec CNT100;
   1:  PR[91,1] = PR[90,1] + 62.627;
   1:  PR[91,2] = PR[90,2] + -21.359;
   1:  PR[91,3] = PR[90,3] + 39.824;
   1:L PR[91] R[100]mm/sec CNT100;
   1:  PR[91,1] = PR[90,1] + 64.586;
   1:  PR[91,2] = PR[90,2] + -21.650;
   1:  PR[91,3] = PR[90,3] + 39.833;
   1:L PR[91] R[100]mm/sec CNT100;
   1:  PR[91,1] = PR[90,1] + 65.060;
   1:  PR[91,2] = PR[90,2] + -21.667;
   1:  PR[91,3] = PR[90,3] + 39.839;
   1:L PR[91] R[100]mm/sec CNT100;
   1:  PR[91,1] = PR[90,1] + 69.373;
   1:  PR[91,2] = PR[90,2] + -21.367;
   1:  PR[91,3] = PR[90,3] + 39.840;
   1:L PR[91] R[100]mm/sec CNT100;
   1:  PR[91,1] = PR[90,1] + 71.350;
   1:  PR[91,2] = PR[90,2] + -21.037;
   1:  PR[91,3] = PR[90,3] + 39.852;
   1:L PR[91] R[100]mm/sec CNT100;
   1:  PR[91,1] = PR[90,1] + 73.854;
   1:  PR[91,2] = PR[90,2] + -20.302;
   1:  PR[91,3] = PR[90,3] + 39.857;
   1:L PR[91] R[100]mm/sec CNT100;
   1:  PR[91,1] = PR[90,1] + 76.784;
   1:  PR[91,2] = PR[90,2] + -19.181;
   1:  PR[91,3] = PR[90,3] + 39.864;
   1:L PR[91] R[100]mm/sec CNT100;
   1:  PR[91,1] = PR[90,1] + 77.938;
   1:  PR[91,2] = PR[90,2] + -18.543;
   1:  PR[91,3] = PR[90,3] + 39.873;
   1:L PR[91] R[100]mm/sec CNT100;
   1:  PR[91,1] = PR[90,1] + 81.256;
   1:  PR[91,2] = PR[90,2] + -16.417;
   1:  PR[91,3] = PR[90,3] + 39.876;
   1:L PR[91] R[100]mm/sec CNT100;
   1:  PR[91,1] = PR[90,1] + 81.539;
   1:  PR[91,2] = PR[90,2] + -16.165;
   1:  PR[91,3] = PR[90,3] + 39.887;
   1:L PR[91] R[100]mm/sec CNT100;
   1:  PR[91,1] = PR[90,1] + 84.672;
   1:  PR[91,2] = PR[90,2] + -13.054;
   1:  PR[91,3] = PR[90,3] + 39.888;
   1:L PR[91] R[100]mm/sec CNT100;
   1:  PR[91,1] = PR[90,1] + 87.040;
   1:  PR[91,2] = PR[90,2] + -9.263;
   1:  PR[91,3] = PR[90,3] + 39.900;
   1:L PR[91] R[100]mm/sec CNT100;
   1:  PR[91,1] = PR[90,1] + 88.500;
   1:  PR[91,2] = PR[90,2] + -5.089;
   1:  PR[91,3] = PR[90,3] + 39.912;
   1:L PR[91] R[100]mm/sec CNT100;
   1:  PR[91,1] = PR[90,1] + 88.994;
   1:  PR[91,2] = PR[90,2] + -0.729;
   1:  PR[91,3] = PR[90,3] + 39.924;
   1:L PR[91] R[100]mm/sec CNT100;
   1:  PR[91,1] = PR[90,1] + 88.500;
   1:  PR[91,2] = PR[90,2] + 3.631;
   1:  PR[91,3] = PR[90,3] + 39.936;
   1:L PR[91] R[100]mm/sec CNT100;
   1:  PR[91,1] = PR[90,1] + 87.040;
   1:  PR[91,2] = PR[90,2] + 7.804;
   1:  PR[91,3] = PR[90,3] + 39.948;
   1:L PR[91] R[100]mm/sec CNT100;
   1:  PR[91,1] = PR[90,1] + 84.672;
   1:  PR[91,2] = PR[90,2] + 11.595;
   1:  PR[91,3] = PR[90,3] + 39.960;
   1:L PR[91] R[100]mm/sec CNT100;
   1:  PR[91,1] = PR[90,1] + 81.539;
   1:  PR[91,2] = PR[90,2] + 14.706;
   1:  PR[91,3] = PR[90,3] + 39.972;
   1:L PR[91] R[100]mm/sec CNT100;
   1:  PR[91,1] = PR[90,1] + 81.256;
   1:  PR[91,2] = PR[90,2] + 14.958;
   1:  PR[91,3] = PR[90,3] + 39.984;
   1:L PR[91] R[100]mm/sec CNT100;
   1:  PR[91,1] = PR[90,1] + 77.939;
   1:  PR[91,2] = PR[90,2] + 17.085;
   1:  PR[91,3] = PR[90,3] + 39.985;
   1:L PR[91] R[100]mm/sec CNT100;
   1:  PR[91,1] = PR[90,1] + 76.784;
   1:  PR[91,2] = PR[90,2] + 17.723;
   1:  PR[91,3] = PR[90,3] + 39.996;
   1:L PR[91] R[100]mm/sec CNT100;
   1:  PR[91,1] = PR[90,1] + 73.855;
   1:  PR[91,2] = PR[90,2] + 18.843;
   1:  PR[91,3] = PR[90,3] + 40.000;
   1:L PR[91] R[100]mm/sec CNT100;
   1:  PR[91,1] = PR[90,1] + 71.351;
   1:  PR[91,2] = PR[90,2] + 19.578;
   1:  PR[91,3] = PR[90,3] + 40.008;
   1:L PR[91] R[100]mm/sec CNT100;
   1:  PR[91,1] = PR[90,1] + 69.373;
   1:  PR[91,2] = PR[90,2] + 19.908;
   1:  PR[91,3] = PR[90,3] + 40.015;
   1:L PR[91] R[100]mm/sec CNT100;
   1:  PR[91,1] = PR[90,1] + 65.061;
   1:  PR[91,2] = PR[90,2] + 20.209;
   1:  PR[91,3] = PR[90,3] + 40.021;
   1:L PR[91] R[100]mm/sec CNT100;
   1:  PR[91,1] = PR[90,1] + 64.587;
   1:  PR[91,2] = PR[90,2] + 20.192;
   1:  PR[91,3] = PR[90,3] + 40.032;
   1:L PR[91] R[100]mm/sec CNT100;
   1:  PR[91,1] = PR[90,1] + 62.627;
   1:  PR[91,2] = PR[90,2] + 19.900;
   1:  PR[91,3] = PR[90,3] + 40.034;
   1:L PR[91] R[100]mm/sec CNT100;
   1:  PR[91,1] = PR[90,1] + 59.327;
   1:  PR[91,2] = PR[90,2] + 19.529;
   1:  PR[91,3] = PR[90,3] + 40.039;
   1:L PR[91] R[100]mm/sec CNT100;
   1:  PR[91,1] = PR[90,1] + 58.031;
   1:  PR[91,2] = PR[90,2] + 19.249;
   1:  PR[91,3] = PR[90,3] + 40.048;
   1:L PR[91] R[100]mm/sec CNT100;
   1:  PR[91,1] = PR[90,1] + 54.681;
   1:  PR[91,2] = PR[90,2] + 18.124;
   1:  PR[91,3] = PR[90,3] + 40.052;
   1:L PR[91] R[100]mm/sec CNT100;
   1:  PR[91,1] = PR[90,1] + 51.281;
   1:  PR[91,2] = PR[90,2] + 16.624;
   1:  PR[91,3] = PR[90,3] + 40.061;
   1:L PR[91] R[100]mm/sec CNT100;
   1:  PR[91,1] = PR[90,1] + 50.557;
   1:  PR[91,2] = PR[90,2] + 16.178;
   1:  PR[91,3] = PR[90,3] + 40.071;
   1:L PR[91] R[100]mm/sec CNT100;
   1:  PR[91,1] = PR[90,1] + 48.787;
   1:  PR[91,2] = PR[90,2] + 14.870;
   1:  PR[91,3] = PR[90,3] + 40.074;
   1:L PR[91] R[100]mm/sec CNT100;
   1:  PR[91,1] = PR[90,1] + 46.675;
   1:  PR[91,2] = PR[90,2] + 13.473;
   1:  PR[91,3] = PR[90,3] + 40.080;
   1:L PR[91] R[100]mm/sec CNT100;
   1:  PR[91,1] = PR[90,1] + 45.788;
   1:  PR[91,2] = PR[90,2] + 12.843;
   1:  PR[91,3] = PR[90,3] + 40.086;
   1:L PR[91] R[100]mm/sec CNT100;
   1:  PR[91,1] = PR[90,1] + 42.110;
   1:  PR[91,2] = PR[90,2] + 8.950;
   1:  PR[91,3] = PR[90,3] + 40.089;
   1:L PR[91] R[100]mm/sec CNT100;
   1:  PR[91,1] = PR[90,1] + 38.518;
   1:  PR[91,2] = PR[90,2] + 13.534;
   1:  PR[91,3] = PR[90,3] + 40.104;
   1:L PR[91] R[100]mm/sec CNT100;
   1:  PR[91,1] = PR[90,1] + 37.865;
   1:  PR[91,2] = PR[90,2] + 14.181;
   1:  PR[91,3] = PR[90,3] + 40.120;
   1:L PR[91] R[100]mm/sec CNT100;
   1:  PR[91,1] = PR[90,1] + 34.261;
   1:  PR[91,2] = PR[90,2] + 16.906;
   1:  PR[91,3] = PR[90,3] + 40.122;
   1:L PR[91] R[100]mm/sec CNT100;
   1:  PR[91,1] = PR[90,1] + 33.989;
   1:  PR[91,2] = PR[90,2] + 17.096;
   1:  PR[91,3] = PR[90,3] + 40.135;
   1:L PR[91] R[100]mm/sec CNT100;
   1:  PR[91,1] = PR[90,1] + 33.372;
   1:  PR[91,2] = PR[90,2] + 17.386;
   1:L PR[91] R[100]mm/sec CNT100;
   1:  PR[91,1] = PR[90,1] + 29.082;
   1:  PR[91,2] = PR[90,2] + 19.144;
   1:  PR[91,3] = PR[90,3] + 40.137;
   1:L PR[91] R[100]mm/sec CNT100;
   1:  PR[91,1] = PR[90,1] + 28.306;
   1:  PR[91,2] = PR[90,2] + 19.295;
   1:  PR[91,3] = PR[90,3] + 40.150;
   1:L PR[91] R[100]mm/sec CNT100;
   1:  PR[91,1] = PR[90,1] + 23.851;
   1:  PR[91,2] = PR[90,2] + 19.880;
   1:  PR[91,3] = PR[90,3] + 40.152;
   1:L PR[91] R[100]mm/sec CNT100;
   1:  PR[91,1] = PR[90,1] + 22.904;
   1:  PR[91,2] = PR[90,2] + 19.826;
   1:  PR[91,3] = PR[90,3] + 40.164;
   1:L PR[91] R[100]mm/sec CNT100;
   1:  PR[91,1] = PR[90,1] + 18.603;
   1:  PR[91,2] = PR[90,2] + 19.269;
   1:  PR[91,3] = PR[90,3] + 40.167;
   1:L PR[91] R[100]mm/sec CNT100;
   1:  PR[91,1] = PR[90,1] + 17.545;
   1:  PR[91,2] = PR[90,2] + 18.934;
   1:  PR[91,3] = PR[90,3] + 40.179;
   1:L PR[91] R[100]mm/sec CNT100;
   1:  PR[91,1] = PR[90,1] + 13.678;
   1:  PR[91,2] = PR[90,2] + 17.350;
   1:  PR[91,3] = PR[90,3] + 40.182;
   1:L PR[91] R[100]mm/sec CNT100;
   1:  PR[91,1] = PR[90,1] + 12.609;
   1:  PR[91,2] = PR[90,2] + 16.684;
   1:  PR[91,3] = PR[90,3] + 40.193;
   1:L PR[91] R[100]mm/sec CNT100;
   1:  PR[91,1] = PR[90,1] + 9.398;
   1:  PR[91,2] = PR[90,2] + 14.245;
   1:  PR[91,3] = PR[90,3] + 40.196;
   1:L PR[91] R[100]mm/sec CNT100;
   1:  PR[91,1] = PR[90,1] + 8.423;
   1:  PR[91,2] = PR[90,2] + 13.220;
   1:  PR[91,3] = PR[90,3] + 40.207;
   1:L PR[91] R[100]mm/sec CNT100;
   1:  PR[91,1] = PR[90,1] + 6.002;
   1:  PR[91,2] = PR[90,2] + 10.091;
   1:  PR[91,3] = PR[90,3] + 40.211;
   1:L PR[91] R[100]mm/sec CNT100;
   1:  PR[91,1] = PR[90,1] + 5.896;
   1:  PR[91,2] = PR[90,2] + 9.926;
   1:  PR[91,3] = PR[90,3] + 40.222;
   1:L PR[91] R[100]mm/sec CNT100;
   1:  PR[91,1] = PR[90,1] + 5.355;
   1:  PR[91,2] = PR[90,2] + 8.893;
   1:L PR[91] R[100]mm/sec CNT100;
   1:  PR[91,1] = PR[90,1] + 4.348;
   1:  PR[91,2] = PR[90,2] + 6.482;
   1:  PR[91,3] = PR[90,3] + 40.226;
   1:L PR[91] R[100]mm/sec CNT100;
   1:  PR[91,1] = PR[90,1] + 3.908;
   1:  PR[91,2] = PR[90,2] + 5.368;
   1:  PR[91,3] = PR[90,3] + 40.233;
   1:L PR[91] R[100]mm/sec CNT100;
   1:  PR[91,1] = PR[90,1] + 3.537;
   1:  PR[91,2] = PR[90,2] + 3.715;
   1:  PR[91,3] = PR[90,3] + 40.236;
   1:L PR[91] R[100]mm/sec CNT100;
   1:  PR[91,1] = PR[90,1] + 0.375;
   1:  PR[91,2] = PR[90,2] + 3.676;
   1:  PR[91,3] = PR[90,3] + 40.241;
   1:L PR[91] R[100]mm/sec CNT100;
   1:  PR[91,1] = PR[90,1] + -0.035;
   1:  PR[91,2] = PR[90,2] + 5.314;
   1:  PR[91,3] = PR[90,3] + 40.249;
   1:L PR[91] R[100]mm/sec CNT100;
   1:  PR[91,1] = PR[90,1] + -1.699;
   1:  PR[91,2] = PR[90,2] + 8.990;
   1:  PR[91,3] = PR[90,3] + 40.254;
   1:L PR[91] R[100]mm/sec CNT100;
   1:  PR[91,1] = PR[90,1] + -1.936;
   1:  PR[91,2] = PR[90,2] + 9.428;
   1:  PR[91,3] = PR[90,3] + 40.265;
   1:L PR[91] R[100]mm/sec CNT100;
   1:  PR[91,1] = PR[90,1] + -4.602;
   1:  PR[91,2] = PR[90,2] + 12.703;
   1:  PR[91,3] = PR[90,3] + 40.266;
   1:L PR[91] R[100]mm/sec CNT100;
   1:  PR[91,1] = PR[90,1] + -4.823;
   1:  PR[91,2] = PR[90,2] + 12.942;
   1:  PR[91,3] = PR[90,3] + 40.278;
   1:L PR[91] R[100]mm/sec CNT100;
   1:  PR[91,1] = PR[90,1] + -7.907;
   1:  PR[91,2] = PR[90,2] + 15.315;
   1:L PR[91] R[100]mm/sec CNT100;
   1:  PR[91,1] = PR[90,1] + -8.529;
   1:  PR[91,2] = PR[90,2] + 15.822;
   1:  PR[91,3] = PR[90,3] + 40.289;
   1:L PR[91] R[100]mm/sec CNT100;
   1:  PR[91,1] = PR[90,1] + -12.584;
   1:  PR[91,2] = PR[90,2] + 17.832;
   1:  PR[91,3] = PR[90,3] + 40.291;
   1:L PR[91] R[100]mm/sec CNT100;
   1:  PR[91,1] = PR[90,1] + -13.033;
   1:  PR[91,2] = PR[90,2] + 17.971;
   1:  PR[91,3] = PR[90,3] + 40.304;
   1:L PR[91] R[100]mm/sec CNT100;
   1:  PR[91,1] = PR[90,1] + -16.934;
   1:  PR[91,2] = PR[90,2] + 18.927;
   1:  PR[91,3] = PR[90,3] + 40.305;
   1:L PR[91] R[100]mm/sec CNT100;
   1:  PR[91,1] = PR[90,1] + -17.995;
   1:  PR[91,2] = PR[90,2] + 19.015;
   1:  PR[91,3] = PR[90,3] + 40.316;
   1:L PR[91] R[100]mm/sec CNT100;
   1:  PR[91,1] = PR[90,1] + -21.404;
   1:  PR[91,2] = PR[90,2] + 19.099;
   1:  PR[91,3] = PR[90,3] + 40.319;
   1:L PR[91] R[100]mm/sec CNT100;
   1:  PR[91,1] = PR[90,1] + -23.008;
   1:  PR[91,2] = PR[90,2] + 18.881;
   1:  PR[91,3] = PR[90,3] + 40.328;
   1:L PR[91] R[100]mm/sec CNT100;
   1:  PR[91,1] = PR[90,1] + -25.792;
   1:  PR[91,2] = PR[90,2] + 18.346;
   1:  PR[91,3] = PR[90,3] + 40.332;
   1:L PR[91] R[100]mm/sec CNT100;
   1:  PR[91,1] = PR[90,1] + -27.769;
   1:  PR[91,2] = PR[90,2] + 17.623;
   1:  PR[91,3] = PR[90,3] + 40.340;
   1:L PR[91] R[100]mm/sec CNT100;
   1:  PR[91,1] = PR[90,1] + -29.903;
   1:  PR[91,2] = PR[90,2] + 16.711;
   1:  PR[91,3] = PR[90,3] + 40.346;
   1:L PR[91] R[100]mm/sec CNT100;
   1:  PR[91,1] = PR[90,1] + -32.013;
   1:  PR[91,2] = PR[90,2] + 15.363;
   1:  PR[91,3] = PR[90,3] + 40.352;
   1:L PR[91] R[100]mm/sec CNT100;
   1:  PR[91,1] = PR[90,1] + -33.550;
   1:  PR[91,2] = PR[90,2] + 14.269;
   1:  PR[91,3] = PR[90,3] + 40.359;
   1:L PR[91] R[100]mm/sec CNT100;
   1:  PR[91,1] = PR[90,1] + -35.535;
   1:  PR[91,2] = PR[90,2] + 12.277;
   1:  PR[91,3] = PR[90,3] + 40.364;
   1:L PR[91] R[100]mm/sec CNT100;
   1:  PR[91,1] = PR[90,1] + -36.573;
   1:  PR[91,2] = PR[90,2] + 11.130;
   1:  PR[91,3] = PR[90,3] + 40.372;
   1:L PR[91] R[100]mm/sec CNT100;
   1:  PR[91,1] = PR[90,1] + -38.277;
   1:  PR[91,2] = PR[90,2] + 8.424;
   1:  PR[91,3] = PR[90,3] + 40.376;
   1:L PR[91] R[100]mm/sec CNT100;
   1:  PR[91,1] = PR[90,1] + -38.454;
   1:  PR[91,2] = PR[90,2] + 8.210;
   1:  PR[91,3] = PR[90,3] + 40.384;
   1:L PR[91] R[100]mm/sec CNT100;
   1:  PR[91,1] = PR[90,1] + -38.674;
   1:  PR[91,2] = PR[90,2] + 7.874;
   1:  PR[91,3] = PR[90,3] + 40.385;
   1:L PR[91] R[100]mm/sec CNT100;
   1:  PR[91,1] = PR[90,1] + -38.918;
   1:  PR[91,2] = PR[90,2] + 7.401;
   1:  PR[91,3] = PR[90,3] + 40.386;
   1:L PR[91] R[100]mm/sec CNT100;
   1:  PR[91,1] = PR[90,1] + -39.698;
   1:  PR[91,2] = PR[90,2] + 5.174;
   1:  PR[91,3] = PR[90,3] + 40.388;
   1:L PR[91] R[100]mm/sec CNT100;
   1:  PR[91,1] = PR[90,1] + -39.794;
   1:  PR[91,2] = PR[90,2] + 5.018;
   1:  PR[91,3] = PR[90,3] + 40.394;
   1:L PR[91] R[100]mm/sec CNT100;
   1:  PR[91,1] = PR[90,1] + -40.058;
   1:  PR[91,2] = PR[90,2] + 4.357;
   1:  PR[91,3] = PR[90,3] + 40.395;
   1:L PR[91] R[100]mm/sec CNT100;
   1:  PR[91,1] = PR[90,1] + -40.648;
   1:  PR[91,2] = PR[90,2] + 1.647;
   1:  PR[91,3] = PR[90,3] + 40.397;
   1:L PR[91] R[100]mm/sec CNT100;
   1:  PR[91,1] = PR[90,1] + -43.844;
   1:  PR[91,2] = PR[90,2] + 1.620;
   1:  PR[91,3] = PR[90,3] + 40.404;
   1:L PR[91] R[100]mm/sec CNT100;
   1:  PR[91,1] = PR[90,1] + -44.437;
   1:  PR[91,2] = PR[90,2] + 4.144;
   1:  PR[91,3] = PR[90,3] + 40.413;
   1:L PR[91] R[100]mm/sec CNT100;
   1:  PR[91,1] = PR[90,1] + -45.376;
   1:  PR[91,2] = PR[90,2] + 6.230;
   1:  PR[91,3] = PR[90,3] + 40.420;
   1:L PR[91] R[100]mm/sec CNT100;
   1:  PR[91,1] = PR[90,1] + -45.953;
   1:  PR[91,2] = PR[90,2] + 7.557;
   1:  PR[91,3] = PR[90,3] + 40.426;
   1:L PR[91] R[100]mm/sec CNT100;
   1:  PR[91,1] = PR[90,1] + -46.287;
   1:  PR[91,2] = PR[90,2] + 8.016;
   1:  PR[91,3] = PR[90,3] + 40.430;
   1:L PR[91] R[100]mm/sec CNT100;
   1:  PR[91,1] = PR[90,1] + -48.091;
   1:  PR[91,2] = PR[90,2] + 10.227;
   1:  PR[91,3] = PR[90,3] + 40.432;
   1:L PR[91] R[100]mm/sec CNT100;
   1:  PR[91,1] = PR[90,1] + -48.983;
   1:  PR[91,2] = PR[90,2] + 11.434;
   1:  PR[91,3] = PR[90,3] + 40.439;
   1:L PR[91] R[100]mm/sec CNT100;
   1:  PR[91,1] = PR[90,1] + -52.557;
   1:  PR[91,2] = PR[90,2] + 14.502;
   1:  PR[91,3] = PR[90,3] + 40.443;
   1:L PR[91] R[100]mm/sec CNT100;
   1:  PR[91,1] = PR[90,1] + -54.553;
   1:  PR[91,2] = PR[90,2] + 15.613;
   1:  PR[91,3] = PR[90,3] + 40.456;
   1:L PR[91] R[100]mm/sec CNT100;
   1:  PR[91,1] = PR[90,1] + -56.754;
   1:  PR[91,2] = PR[90,2] + 16.812;
   1:  PR[91,3] = PR[90,3] + 40.462;
   1:L PR[91] R[100]mm/sec CNT100;
   1:  PR[91,1] = PR[90,1] + -61.370;
   1:  PR[91,2] = PR[90,2] + 18.300;
   1:  PR[91,3] = PR[90,3] + 40.469;
   1:L PR[91] R[100]mm/sec CNT100;
   1:  PR[91,1] = PR[90,1] + -62.381;
   1:  PR[91,2] = PR[90,2] + 18.428;
   1:  PR[91,3] = PR[90,3] + 40.482;
   1:L PR[91] R[100]mm/sec CNT100;
   1:  PR[91,1] = PR[90,1] + -65.992;
   1:  PR[91,2] = PR[90,2] + 18.957;
   1:  PR[91,3] = PR[90,3] + 40.485;
   1:L PR[91] R[100]mm/sec CNT100 TB   .50sec,CALL END_PUD;
   1:  DO[117:Laser Start]=OFF;
   1:  PR[92] = PR[91];
   1:  PR[92,3] = PR[92,3] + 50;
   1:J PR[92] 10% FINE;
   1:  WAIT   5.00(sec);
   1:  DO[119:Gas]=OFF;
   1:  CALL HOME_ALL;
/POS
/END
